Staubli VAL3: ros2_server.dtx

public sio siSocketControl = {link=UdpSocket\fuzzyudp}
public bool bIsOverrun = true
mdesc mMdesc = {blend=off}
public num nErrorCode
public num nInError
public num nOverruns
